PROGRAM P06_WickFeeder
VAR_INPUT
	IbWickFeederDragHomingSensor 			  	: BOOL;				// Czujnik bazowania
	IbWickFeederDragUpSensor 			 	  	: BOOL;				// Czujnik
	IbWickFeederDragDownSensor 				 	: BOOL;				// Czujnik
	IbWickFeederDragLeadBefore1UpSensor 		: BOOL;				// Czujnik
	IbWickFeederDownSensor1 					: BOOL;								
	IbWheelLevelSensor								: BOOL;			

	IbWheelSensor									: BOOL;			//Czujnik zapełnienia rękawa
	IbQueFullAfterWheelSensor						: BOOL;			
	IbQueFullSensor									: BOOL;			//Czujnik zapełnienia rękawa
	IbWickAtPipe									: BOOL;			//Czujnik na końcu rękawa
	IbSeparatorPos1									: BOOL;			//Separator nad torem 1
	IbSeparatorPos2									: BOOL;			//Separator nad torem 2
	IbQueFullAtSleve1								: BOOL;			//Czujnik zapełnienia rękawa 1
	IbQueFullAtSleve2								: BOOL;			//Czujnik zapełnienia rękawa 2
	IbWickAtSleve1									: BOOL;			//Czujnik na końcu rękawa 1
	IbWickAtSleve2									: BOOL;			//Czujnik na końcu rękawa 2
	IbSleve1SeparatorOut							: BOOL;			//Separator nad butelką
	IbSleve2SeparatorOut							: BOOL;			//Separator nad butelką
	IbHammer1Up										: BOOL;			//Wbijak pozycja górna
	IbHammer1Down									: BOOL;			//Wbijak pozycja dolna
	IbHammer2Up										: BOOL;			//Wbijak pozycja górna
	IbHammer2Down									: BOOL;			//Wbijak pozycja dolna
	IbFormPositioningHide1							: BOOL; 
	IbFormPositioningHide2							: BOOL;

	QbStopper1										: BOOL;			//Stoper przed separatorem
	QbStopper2										: BOOL;			//Stoper przed separatorem
	QbSeparator1									: BOOL;			//Separator nad torem 1
	QbSeparator2									: BOOL;			//Separator nad torem 2
	QbSleve1SeparatorActIn							: BOOL;			//Separator pod rękawem
	QbSleve1SeparatorActOut							: BOOL;			//Separator nad butelką
	QbSleve2SeparatorActIn							: BOOL;			//Separator pod rękawem
	QbSleve2SeparatorActOut							: BOOL;			//Separator nad butelką
	QbHammer1										: BOOL;			//Wbijak 
	QbHammer2										: BOOL;			//Wbijak
	QbBlow1											: BOOL;
	QbSleeveBlow									: BOOL;
	QbFormPositioning								: BOOL;  		


	bMovetoEndPositionWickFeeder				: BOOL;	
	QbWickFeederDragActuator                  	: BOOL;				// Siłownikiem przeciągania (1 faza)					

	
	QbWickFeederSorterEngine					AT %Q*	: BOOL; 					// Wyjście silnikiem sortera
	QbWickFeederSorterAir 						AT %Q*	: BOOL; 					// Wyjście sterujące szybkim zaworem wydmuchu
	QbWickFeederSorterAir2 						AT %Q*	: BOOL; 					// Wyjście sterujące szybkim zaworem wydmuchu
	
	IbFuseWickFeederSorterEngineOK			AT %I*	: BOOL;					//Bezpiecznik silnika sortera OK

	QnWickFeederSorterVelocitySV 			AT %Q*	: UDINT; 		// Nastawa prędkości
	InWickFeederSorterVelocityCV 			AT %I*	: UDINT;		
	InWickFeederSorterSTW 					AT %I*	: UINT; 		// Statusword transportera wejściowo wyjściowego
	QnWickFeederSorterCTW 					AT %Q*	: UINT;  		// Controlword transportera we/wy
                                                  		
	TimerWickFeederSorterEnable						: TOF;
	tonWickFeederSorterEnable						: TON;
	
END_VAR
VAR
	//Podajnik knotów
	fbWickFeederSt									: FB_WickFeederStation; 				// Blok sterowania
	eWickFeederState								: E_Station; 							// Stan pracy podajnika platynek			
	eWickFeederRunningState							: E_WickFeederState; 					// Stan pracy podajnika platynek
	fbWickFeederState								: FB_State; 


	QbWickFeeder_HeightMotorUp 				AT %Q*	: BOOL;									// Sterowanie silnikiem podnosnika stacji w górę 
	QbWickFeeder_HeightMotorDown 			AT %Q*	: BOOL;									//Sterowanie silnikiem podnosnika stacji w dół
	
	
	IbWickFeeder2DownSensor1 				AT %I*	: BOOL;								
	IbWickFeederHeightEncoderSetCDone		AT %I*	: BOOL;	
	IudiWickFeederHeightEncoderCV         	AT %I*	: UDINT; 	
	QbWickFeederHeightEncoderSetC 			AT %Q*	: BOOL;		
	QudiWickFeederHeightEncoderSetCV       	AT %Q*	: UDINT; 	
	
	tofWickFeederEnable								: TOF;
	tonWickFeederEnable								: TON;
	rtEnable										: R_TRIG;

	bSimulation										: BOOL;
	
	bWickFeederWarning1								: BOOL;
	bWickFeederWarning2								: BOOL;
	
	//PRZECIAGANIE
	eWickFeederDragStation							: E_Station;
	eWickFeederDragRunningStation					: E_DragStationState;
	fbWickFeederDragStation							: FB_FormsDragStepper;

	tofWickFeederDragStationEnable					: TOF;	
	
	//WEJSCIA I WYJSCIA SPRZETOWE
	QbWickFeederDragLeadBefore1Actuator        		: BOOL;				// Siłownikiem prowadzenia przed 1(1 faza)
	QbWickFeederDragLeadBefore2Actuator        		: BOOL;				// Siłownikiem prowadzenia przed 1(1 faza)
	


	bTestManual										: BOOL;	
	bWickFeederSorterRunTest						: BOOL;
	bWickFeeder1RunTest								: BOOL;
	bWickFeeder2RunTest								: BOOL;
	tonQbSleve1SeparatorActIn						:TON;
	tonQbSleve2SeparatorActIn						:TON;	
END_VAR


ACT_Limits();
ACT_WickFeederStation();
ACT_WickFeederDragStation();
aWickFeederWarnings();

//GENEROWANIE STANU STACJI DO WIZKI
tonQbSleve1SeparatorActIn	(IN:=QbSleve1SeparatorActIn, PT:=T#100MS);
tonQbSleve2SeparatorActIn	(IN:=QbSleve2SeparatorActIn, PT:=T#100MS);

(* BAZOWANIE - ZMIAN*)
tonWickFeederEnable(IN := fbWickFeederSt.bEnable, PT := T#2S); (*Dodany ton bo Wizka zjebnie wgrywa zmienne, najpierw włacza Enabla a potem dopiero wybiera recepture*)
rtEnable(CLK := tonWickFeederEnable.Q, Q=>);
IF rtEnable.Q AND (P00_PackML.fbPMLAuto.ePMLState = Tc3_PackML.E_PMLState.ePMLState_IDLE OR 
   P00_PackML.fbPMLAuto.ePMLState = Tc3_PackML.E_PMLState.ePMLState_EXECUTE) THEN
    VIS.bWickFeederHeightSet 		:= TRUE;
ELSIF fbWickFeederst.eState = E_Station.eHomingDone OR VIS.bErrorOccure THEN
    VIS.bWickFeederHeightSet 		:= FALSE;
END_IF
(*KONIEC BAZOWANIE - ZMIANA*)

//PRZEPISYWANIE POMIARÓW

//SYMULACJA CZUJNIKÓW IGLIC

//Opoznienie wyłączanie enabla
tofWickFeederEnable(IN:= bWickFeederEnable, PT:=T#2S);

//KASOWANIE ROZKAZÓW CYKLI
IF fbWickFeederst.bCycleDone1 AND GVL.bManualMode THEN
	VIS.bWickFeeder1Run 			:= FALSE;
END_IF
IF fbWickFeederst.bCycleDone2 AND GVL.bManualMode THEN
	VIS.bWickFeeder2Run 			:= FALSE;
END_IF

IF bSimulation THEN
	IF fbWickFeederSt.eRunningState1 = E_WickFeederState.eReady  THEN
		VIS.bWickFeeder1Run	:= TRUE;
	END_IF
	IF fbWickFeederSt.eRunningState2 = E_WickFeederState.eReady  THEN
		VIS.bWickFeeder2Run	:= TRUE;
	END_IF	
	

	IF fbWickFeederSt.bCycleDone1 THEN		
		VIS.bWickFeeder1Run 		:= FALSE;	
	END_IF
	IF fbWickFeederSt.bCycleDone2 THEN		
		VIS.bWickFeeder2Run 		:= FALSE;	
	END_IF
END_IF

//Przeciąganie
tofWickFeederDragStationEnable(IN:= bWickFeederDragingStationEnable, PT:= T#2S);


////ZBIORNIK I SORTER KNOTÓW
aWickFeederSorterWarnings();
QbWickFeederSorterAir2 :=	QbWickFeederSorterEngine OR QbWickFeederSorterAir; //Dodatkowy przedmuch


(*Opoznienie wyłączanie enabla*)

ACTION ACT_Limits:
(*
Nazwa:			aSetRecipe
Opis:			Zapisywanie zmiennych gdy mają wartość 0 
Wersja:			v0.1
Data:			2022-06-22
Autor:			DP
Urzadzenia:		
Konfiguracja:	
Info:
- zabezpieczenie przed recepturami które nie mają tych parametrów i jest w nich wartość 0
*)

IF 	VIS.lrWickFeedingDragingStationStartPosition		= 0		THEN	VIS.lrWickFeedingDragingStationStartPosition		:=	8;		END_IF;
IF 	VIS.lrWickFeedingDragingStationEndPosition		= 0		THEN	VIS.lrWickFeedingDragingStationEndPosition		:=	138;	END_IF;
END_ACTION

ACTION ACT_WickFeederDragStation:
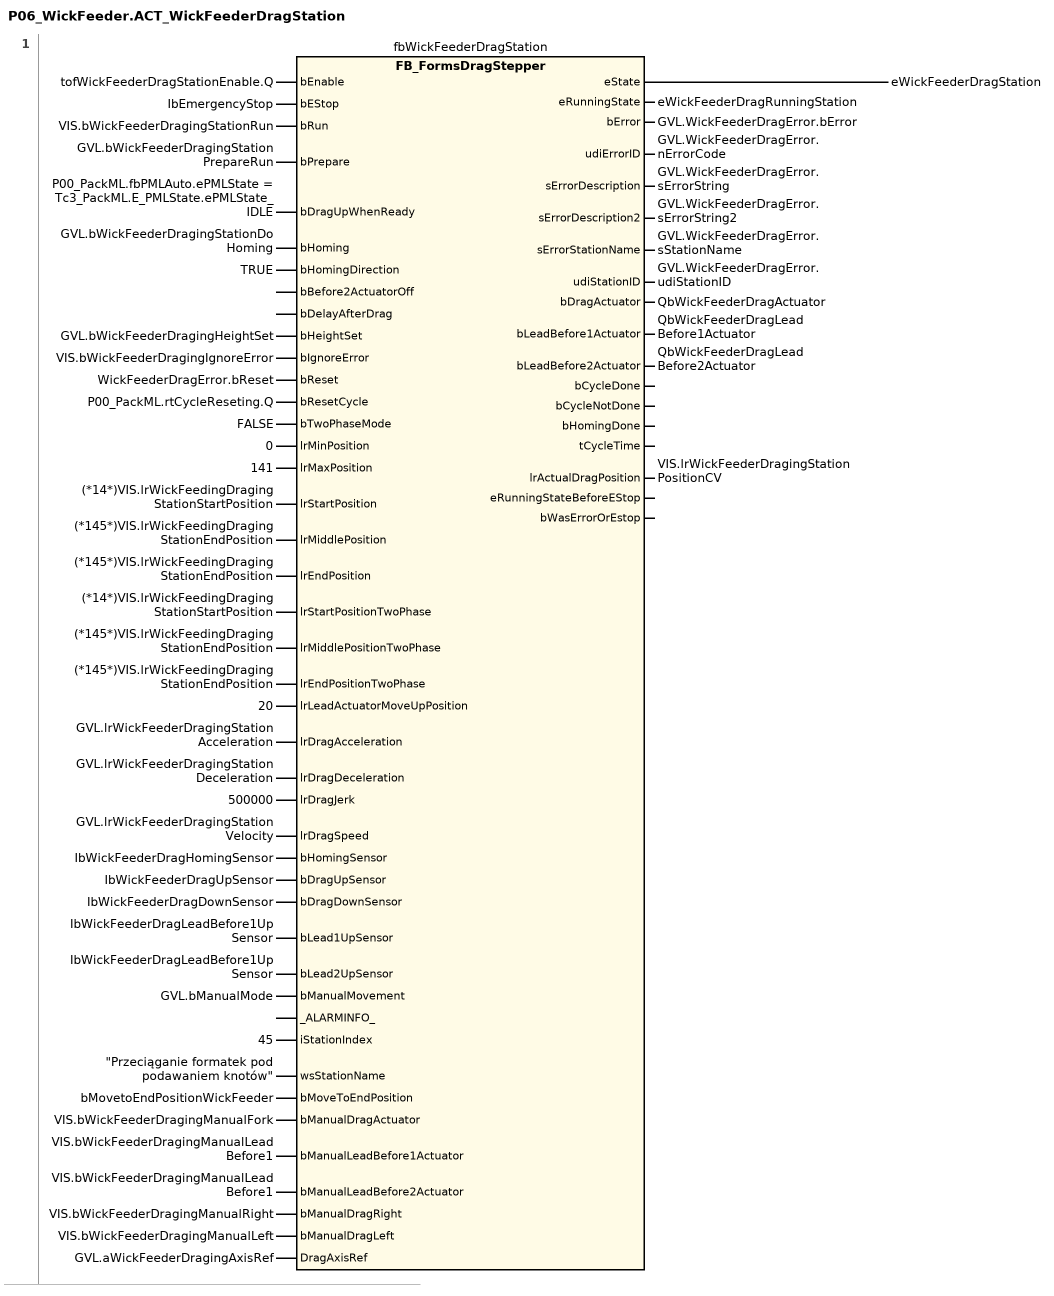
// NETWORK 1
fbWickFeederDragStation(
    bEnable := tofWickFeederDragStationEnable.Q,
    bEStop := IbEmergencyStop,
    bRun := VIS.bWickFeederDragingStationRun,
    bPrepare := GVL.bWickFeederDragingStationPrepareRun,
    bDragUpWhenReady := P00_PackML.fbPMLAuto.ePMLState = Tc3_PackML.E_PMLState.ePMLState_IDLE,
    bHoming := GVL.bWickFeederDragingStationDoHoming,
    bHomingDirection := TRUE,
    bHeightSet := GVL.bWickFeederDragingHeightSet,
    bIgnoreError := VIS.bWickFeederDragingIgnoreError,
    bReset := WickFeederDragError.bReset,
    bResetCycle := P00_PackML.rtCycleReseting.Q,
    bTwoPhaseMode := FALSE,
    lrMinPosition := 0,
    lrMaxPosition := 141,
    lrStartPosition := (*14*)VIS.lrWickFeedingDragingStationStartPosition,
    lrMiddlePosition := (*145*)VIS.lrWickFeedingDragingStationEndPosition,
    lrEndPosition := (*145*)VIS.lrWickFeedingDragingStationEndPosition,
    lrStartPositionTwoPhase := (*14*)VIS.lrWickFeedingDragingStationStartPosition,
    lrMiddlePositionTwoPhase := (*145*)VIS.lrWickFeedingDragingStationEndPosition,
    lrEndPositionTwoPhase := (*145*)VIS.lrWickFeedingDragingStationEndPosition,
    lrLeadActuatorMoveUpPosition := 20,
    lrDragAcceleration := GVL.lrWickFeederDragingStationAcceleration,
    lrDragDeceleration := GVL.lrWickFeederDragingStationDeceleration,
    lrDragJerk := 500000,
    lrDragSpeed := GVL.lrWickFeederDragingStationVelocity,
    bHomingSensor := IbWickFeederDragHomingSensor,
    bDragUpSensor := IbWickFeederDragUpSensor,
    bDragDownSensor := IbWickFeederDragDownSensor,
    bLead1UpSensor := IbWickFeederDragLeadBefore1UpSensor,
    bLead2UpSensor := IbWickFeederDragLeadBefore1UpSensor,
    bManualMovement := GVL.bManualMode,
    iStationIndex := 45,
    wsStationName := "Przeciąganie formatek pod podawaniem knotów",
    bMoveToEndPosition := bMovetoEndPositionWickFeeder,
    bManualDragActuator := VIS.bWickFeederDragingManualFork,
    bManualLeadBefore1Actuator := VIS.bWickFeederDragingManualLeadBefore1,
    bManualLeadBefore2Actuator := VIS.bWickFeederDragingManualLeadBefore1,
    bManualDragRight := VIS.bWickFeederDragingManualRight,
    bManualDragLeft := VIS.bWickFeederDragingManualLeft,
    DragAxisRef := GVL.aWickFeederDragingAxisRef,
    eRunningState => eWickFeederDragRunningStation,
    bError => GVL.WickFeederDragError.bError,
    udiErrorID => GVL.WickFeederDragError.nErrorCode,
    sErrorDescription => GVL.WickFeederDragError.sErrorString,
    sErrorDescription2 => GVL.WickFeederDragError.sErrorString2,
    sErrorStationName => GVL.WickFeederDragError.sStationName,
    udiStationID => GVL.WickFeederDragError.udiStationID,
    bDragActuator => QbWickFeederDragActuator,
    bLeadBefore1Actuator => QbWickFeederDragLeadBefore1Actuator,
    bLeadBefore2Actuator => QbWickFeederDragLeadBefore2Actuator,
    lrActualDragPosition => VIS.lrWickFeederDragingStationPositionCV); // FB_FormsDragStepper
eWickFeederDragStation := fbWickFeederDragStation.eState;
END_ACTION

ACTION ACT_WickFeederStation:
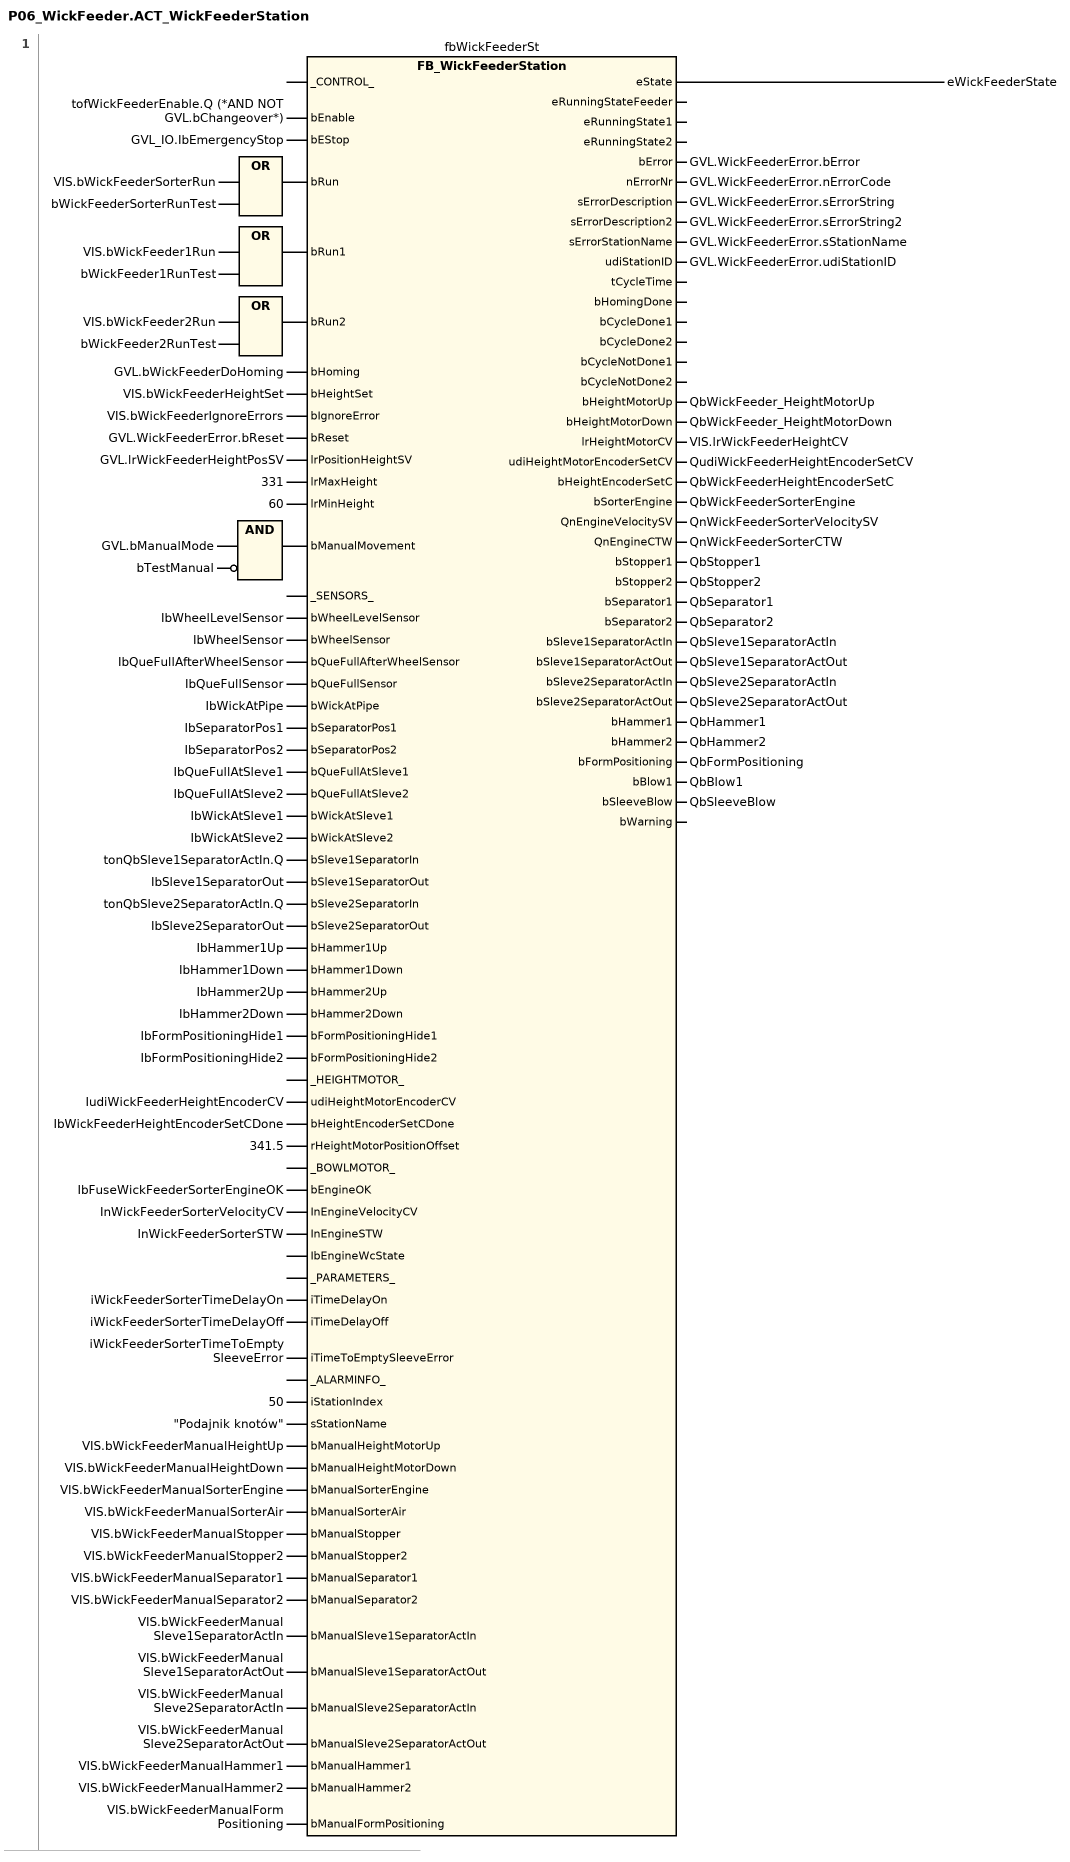
// NETWORK 1
fbWickFeederSt(
    bEnable := tofWickFeederEnable.Q (*AND NOT GVL.bChangeover*),
    bEStop := GVL_IO.IbEmergencyStop,
    bRun := VIS.bWickFeederSorterRun OR bWickFeederSorterRunTest,
    bRun1 := VIS.bWickFeeder1Run OR bWickFeeder1RunTest,
    bRun2 := VIS.bWickFeeder2Run OR bWickFeeder2RunTest,
    bHoming := GVL.bWickFeederDoHoming,
    bHeightSet := VIS.bWickFeederHeightSet,
    bIgnoreError := VIS.bWickFeederIgnoreErrors,
    bReset := GVL.WickFeederError.bReset,
    lrPositionHeightSV := GVL.lrWickFeederHeightPosSV,
    lrMaxHeight := 331,
    lrMinHeight := 60,
    bManualMovement := GVL.bManualMode AND NOT bTestManual,
    bWheelLevelSensor := IbWheelLevelSensor,
    bWheelSensor := IbWheelSensor,
    bQueFullAfterWheelSensor := IbQueFullAfterWheelSensor,
    bQueFullSensor := IbQueFullSensor,
    bWickAtPipe := IbWickAtPipe,
    bSeparatorPos1 := IbSeparatorPos1,
    bSeparatorPos2 := IbSeparatorPos2,
    bQueFullAtSleve1 := IbQueFullAtSleve1,
    bQueFullAtSleve2 := IbQueFullAtSleve2,
    bWickAtSleve1 := IbWickAtSleve1,
    bWickAtSleve2 := IbWickAtSleve2,
    bSleve1SeparatorIn := tonQbSleve1SeparatorActIn.Q,
    bSleve1SeparatorOut := IbSleve1SeparatorOut,
    bSleve2SeparatorIn := tonQbSleve2SeparatorActIn.Q,
    bSleve2SeparatorOut := IbSleve2SeparatorOut,
    bHammer1Up := IbHammer1Up,
    bHammer1Down := IbHammer1Down,
    bHammer2Up := IbHammer2Up,
    bHammer2Down := IbHammer2Down,
    bFormPositioningHide1 := IbFormPositioningHide1,
    bFormPositioningHide2 := IbFormPositioningHide2,
    udiHeightMotorEncoderCV := IudiWickFeederHeightEncoderCV,
    bHeightEncoderSetCDone := IbWickFeederHeightEncoderSetCDone,
    rHeightMotorPositionOffset := 341.5,
    bEngineOK := IbFuseWickFeederSorterEngineOK,
    InEngineVelocityCV := InWickFeederSorterVelocityCV,
    InEngineSTW := InWickFeederSorterSTW,
    iTimeDelayOn := iWickFeederSorterTimeDelayOn,
    iTimeDelayOff := iWickFeederSorterTimeDelayOff,
    iTimeToEmptySleeveError := iWickFeederSorterTimeToEmptySleeveError,
    iStationIndex := 50,
    sStationName := "Podajnik knotów",
    bManualHeightMotorUp := VIS.bWickFeederManualHeightUp,
    bManualHeightMotorDown := VIS.bWickFeederManualHeightDown,
    bManualSorterEngine := VIS.bWickFeederManualSorterEngine,
    bManualSorterAir := VIS.bWickFeederManualSorterAir,
    bManualStopper := VIS.bWickFeederManualStopper,
    bManualStopper2 := VIS.bWickFeederManualStopper2,
    bManualSeparator1 := VIS.bWickFeederManualSeparator1,
    bManualSeparator2 := VIS.bWickFeederManualSeparator2,
    bManualSleve1SeparatorActIn := VIS.bWickFeederManualSleve1SeparatorActIn,
    bManualSleve1SeparatorActOut := VIS.bWickFeederManualSleve1SeparatorActOut,
    bManualSleve2SeparatorActIn := VIS.bWickFeederManualSleve2SeparatorActIn,
    bManualSleve2SeparatorActOut := VIS.bWickFeederManualSleve2SeparatorActOut,
    bManualHammer1 := VIS.bWickFeederManualHammer1,
    bManualHammer2 := VIS.bWickFeederManualHammer2,
    bManualFormPositioning := VIS.bWickFeederManualFormPositioning,
    bError => GVL.WickFeederError.bError,
    nErrorNr => GVL.WickFeederError.nErrorCode,
    sErrorDescription => GVL.WickFeederError.sErrorString,
    sErrorDescription2 => GVL.WickFeederError.sErrorString2,
    sErrorStationName => GVL.WickFeederError.sStationName,
    udiStationID => GVL.WickFeederError.udiStationID,
    bHeightMotorUp => QbWickFeeder_HeightMotorUp,
    bHeightMotorDown => QbWickFeeder_HeightMotorDown,
    lrHeightMotorCV => VIS.lrWickFeederHeightCV,
    udiHeightMotorEncoderSetCV => QudiWickFeederHeightEncoderSetCV,
    bHeightEncoderSetC => QbWickFeederHeightEncoderSetC,
    bSorterEngine => QbWickFeederSorterEngine,
    QnEngineVelocitySV => QnWickFeederSorterVelocitySV,
    QnEngineCTW => QnWickFeederSorterCTW,
    bStopper1 => QbStopper1,
    bStopper2 => QbStopper2,
    bSeparator1 => QbSeparator1,
    bSeparator2 => QbSeparator2,
    bSleve1SeparatorActIn => QbSleve1SeparatorActIn,
    bSleve1SeparatorActOut => QbSleve1SeparatorActOut,
    bSleve2SeparatorActIn => QbSleve2SeparatorActIn,
    bSleve2SeparatorActOut => QbSleve2SeparatorActOut,
    bHammer1 => QbHammer1,
    bHammer2 => QbHammer2,
    bFormPositioning => QbFormPositioning,
    bBlow1 => QbBlow1,
    bSleeveBlow => QbSleeveBlow); // FB_WickFeederStation
eWickFeederState := fbWickFeederSt.eState;
END_ACTION

ACTION aWickFeederSorterWarnings:
// Sorter nasadek
(*
IF fbWickFeederSt.bWarning1 AND NOT WickFeederSorterWarning[0].bWarning THEN
	WickFeederSorterWarning[0].bWarning										:= TRUE;
	WickFeederSorterWarning[0].udiWarningCode									:= 33;	
	WickFeederSorterWarning[0].sDescription									:= 'Podajnik knotów | Niski poziom wkładów';
ELSIF NOT fbWickFeederSt.bWarning1  AND WickFeederSorterWarning[0].bAcknowledge THEN
	WickFeederSorterWarning[0].bWarning										:= FALSE;
	WickFeederSorterWarning[0].bAcknowledge									:= FALSE;
	VIS.uliWarningAcknowledge.14 										:= FALSE;
ELSIF WickFeederSorterWarning[0].bAcknowledge THEN
	WickFeederSorterWarning[0].bAcknowledge									:= TRUE;
END_IF*)
END_ACTION

ACTION aWickFeederWarnings:

//Warning 0
LidFeederWarning[0].sDescription:='Podajnik knotów | Niski poziom';
IF P06_WickFeeder.fbWickFeederSt.bWarning AND NOT LidFeederWarning[0].bWarning AND bWickFeederEnable THEN
	LidFeederWarning[0].bWarning:=TRUE;
ELSIF NOT P06_WickFeeder.fbWickFeederSt.bWarning  AND LidFeederWarning[0].bAcknowledge THEN
	LidFeederWarning[0].bWarning		:=	FALSE;
	LidFeederWarning[0].bAcknowledge	:=	FALSE;
	VIS.uliWarningOccure.39				:=	FALSE;
ELSIF LidFeederWarning[0].bAcknowledge THEN
	LidFeederWarning[0].bAcknowledge	:=	TRUE;
END_IF

//Warning 1
(*WickFeederWarning[1].sDescription:='Podajnik knotów 2 | Brak knotów w zasobniku';
IF bWickFeederWarning2 AND NOT WickFeederWarning[1].bWarning AND bWickFeederEnable THEN
	WickFeederWarning[1].bWarning:=TRUE;
ELSIF NOT bWickFeederWarning2 AND WickFeederWarning[1].bAcknowledge THEN
	WickFeederWarning[1].bWarning		:=	FALSE;
	WickFeederWarning[1].bAcknowledge	:=	FALSE;
	VIS.uliWarningOccure.40				:=	FALSE;
ELSIF WickFeederWarning[1].bAcknowledge THEN
	WickFeederWarning[1].bAcknowledge	:=	TRUE;
END_IF*)
END_ACTION

END_PROGRAM

(* stored: Version 1.2.0.0, ProductVersion 3.1.4026.13, FileIdentifier 3155f1880f4660669d440b652be1e8df88de855b, FileSignature 764fab147b24eed46103b610f63ae49467430e66c029f92d7aa8e8efcba4bc36af698ebf03e0f74b9801a3ec804940cdef86c4196803c0c36af2a9a99dd0dc52f43d7acecee66f53479495205155cec2e11cff0bc23ce4a51234e1a7f61fbf7a3f0f6079eac21a36623fb4f709b2ae4503c539d86ef5d1f55d69f2cc47ba8091a7cb856e7a2b7d6b2e97f04efb6d7d2bd488318daa59c40d9881b8e9eb58024fb9d8774904326c7cce254fdf922f76d55a5d3762e5fc4f4aaca074d8979d7d3d4a4a9bc3aa270ef60fa1915aadba93818fbb86c40ec495d27be2c7ba9f30846090c9f33ce2dd3ebfad3e9dd6f438f9577c58e778f55c7e21de2eadcdcfdaa65c
   POU P06_WickFeeder: Id {59c2b4d0-c718-4a27-af42-66a4f6bb5cca}, SpecialFunc None
   Action ACT_Limits: Id {44093b15-4c19-405d-aaed-7334991f13d9}
   Action ACT_WickFeederDragStation: Id {afbd28a6-dce1-455a-b047-bc4a2411e245}
   Action ACT_WickFeederStation: Id {aefd363d-a56b-4549-8072-46a1371755be}
   Action aWickFeederSorterWarnings: Id {4a1be6bd-12c8-4b31-9c45-5e627d04cdc8}
   Action aWickFeederWarnings: Id {c76a4ced-429c-4830-835d-ca34185440b2} *)
